{attribute 'GeneratedUsingTerminal: EL1809-0000-0018'}
{attribute addProperty BoxType "EL1809-0000-0018"}
{attribute addProperty Id "Channel_1AT %I*Channel_830843C11Channel_2AT %I*Channel_830843C11Channel_3AT %I*Channel_830843C11Channel_4AT %I*Channel_830843C11Channel_5AT %I*Channel_830843C11Channel_6AT %I*Channel_830843C11Channel_7AT %I*Channel_830843C11Channel_8AT %I*Channel_830843C11Channel_9AT %I*Channel_830843C11Channel_10AT %I*Channel_830843C11Channel_11AT %I*Channel_830843C11Channel_12AT %I*Channel_830843C11Channel_13AT %I*Channel_830843C11Channel_14AT %I*Channel_830843C11Channel_15AT %I*Channel_830843C11Channel_16AT %I*Channel_830843C11WcStateAT %I*WcState_9091E0EB2InfoDataAT %I*InfoData_6F19DB2B2"}
{attribute addProperty CRC "840269053"}
{attribute addProperty Size "20"}
TYPE EL1809_32157CFD EXTENDS TcoIo.EtcSlaveTerminalBase_947E5A46 :
STRUCT
	{attribute addProperty Name "Channel_1"}
	Channel_1 : TcoIo.Channel_830843C1;
	{attribute addProperty Name "Channel_2"}
	Channel_2 : TcoIo.Channel_830843C1;
	{attribute addProperty Name "Channel_3"}
	Channel_3 : TcoIo.Channel_830843C1;
	{attribute addProperty Name "Channel_4"}
	Channel_4 : TcoIo.Channel_830843C1;
	{attribute addProperty Name "Channel_5"}
	Channel_5 : TcoIo.Channel_830843C1;
	{attribute addProperty Name "Channel_6"}
	Channel_6 : TcoIo.Channel_830843C1;
	{attribute addProperty Name "Channel_7"}
	Channel_7 : TcoIo.Channel_830843C1;
	{attribute addProperty Name "Channel_8"}
	Channel_8 : TcoIo.Channel_830843C1;
	{attribute addProperty Name "Channel_9"}
	Channel_9 : TcoIo.Channel_830843C1;
	{attribute addProperty Name "Channel_10"}
	Channel_10 : TcoIo.Channel_830843C1;
	{attribute addProperty Name "Channel_11"}
	Channel_11 : TcoIo.Channel_830843C1;
	{attribute addProperty Name "Channel_12"}
	Channel_12 : TcoIo.Channel_830843C1;
	{attribute addProperty Name "Channel_13"}
	Channel_13 : TcoIo.Channel_830843C1;
	{attribute addProperty Name "Channel_14"}
	Channel_14 : TcoIo.Channel_830843C1;
	{attribute addProperty Name "Channel_15"}
	Channel_15 : TcoIo.Channel_830843C1;
	{attribute addProperty Name "Channel_16"}
	Channel_16 : TcoIo.Channel_830843C1;
	{attribute addProperty Name "WcState"}
	WcState : WcState_9091E0EB;
	{attribute addProperty Name "InfoData"}
	InfoData : InfoData_6F19DB2B;
END_STRUCT
END_TYPE

(* stored: Version 1.2.0.0, ProductVersion 3.1.4024.9
   DUT EL1809_32157CFD: Id {189eb9ae-9105-4644-9d16-64d7d962b804} *)
